PROGRAM MAIN_1
VAR
END_VAR

END_PROGRAM

(* stored: Version 1.1.0.1, ProductVersion 3.1.4024.11
   POU MAIN_1: Id {94a3cf28-c82f-432b-98ee-a1011d16688e}, SpecialFunc None *)
